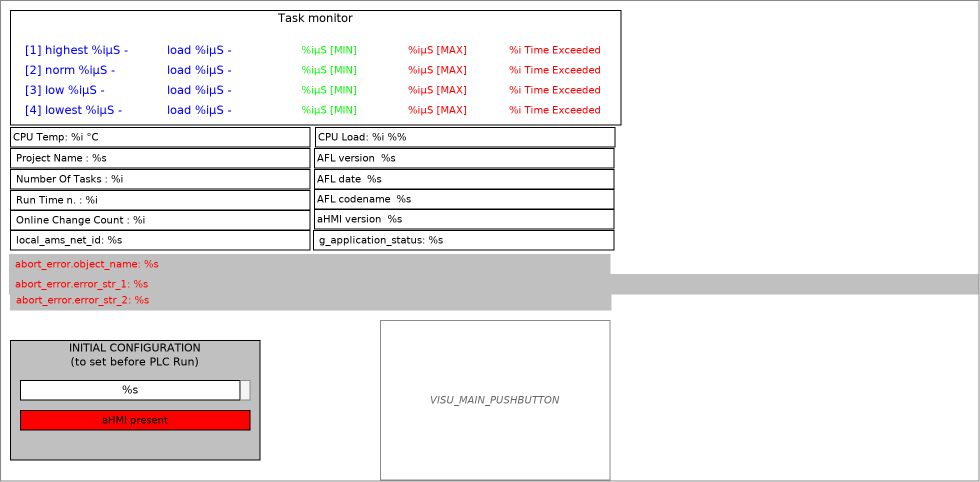
VISUALIZATION VISU_MAIN  // 980x482
    Rectangle (10,10 611x115), "Task monitor"
    Rectangle (9,254 601x20), "abort_error.object_name: %s", text variable: abort_error.object_name
    Rectangle (9,274 969x20), "abort_error.error_str_1: %s", text variable: abort_error.error_str_1
    Rectangle (10,290 601x20), "abort_error.error_str_2: %s", text variable: abort_error.error_str_2
    Rectangle (10,230 300x20), "local_ams_net_id: %s", text variable: local_ams_net_id
    Rectangle (313,230 301x20), "g_application_status: %s", text variable: Application_Common.g_application_status
    Rectangle (22,40 130x20), "[1] highest %iµS -", text variable: afl_tasks[1].cycle_us
    Rectangle (22,60 130x20), "[2] norm %iµS -", text variable: afl_tasks[2].cycle_us
    Rectangle (22,80 130x20), "[3] low %iµS -", text variable: afl_tasks[3].cycle_us
    Rectangle (22,100 130x20), "[4] lowest %iµS -", text variable: afl_tasks[4].cycle_us
    Rectangle (164,100 100x20), "load %iµS -", text variable: afl_tasks[4].task_profiler_data.AverageExecTime
    Rectangle (164,80 100x20), "load %iµS -", text variable: afl_tasks[3].task_profiler_data.AverageExecTime
    Rectangle (164,60 100x20), "load %iµS -", text variable: afl_tasks[2].task_profiler_data.AverageExecTime
    Rectangle (164,40 100x20), "load %iµS -", text variable: afl_tasks[1].task_profiler_data.AverageExecTime
    Rectangle (380,40 90x20), "%iµS [MAX]", text variable: afl_tasks[1].task_profiler_data.MaxExecTime
    Rectangle (380,60 90x20), "%iµS [MAX]", text variable: afl_tasks[2].task_profiler_data.MaxExecTime
    Rectangle (380,80 90x20), "%iµS [MAX]", text variable: afl_tasks[2].task_profiler_data.MaxExecTime
    Rectangle (380,100 90x20), "%iµS [MAX]", text variable: afl_tasks[4].task_profiler_data.MaxExecTime
    Rectangle (10,148 300x20), "Project Name : %s", text variable: SystemInfo.projectName
    Rectangle (10,169 300x20), "Number Of Tasks : %i", text variable: SystemInfo.numberOfTasks
    Rectangle (10,190 300x20), "Run Time n. : %i", text variable: SystemInfo.runTimeNo
    Rectangle (10,210 300x20), "Online Change Count : %i", text variable: SystemInfo.onlineChangeCount
    Rectangle (250,100 110x20), "%iµS [MIN]", text variable: afl_tasks[4].task_profiler_data.MinExecTime
    Rectangle (250,80 110x20), "%iµS [MIN]", text variable: afl_tasks[3].task_profiler_data.MinExecTime
    Rectangle (250,60 110x20), "%iµS [MIN]", text variable: afl_tasks[2].task_profiler_data.MinExecTime
    Rectangle (250,40 110x20), "%iµS [MIN]", text variable: afl_tasks[1].task_profiler_data.MinExecTime
    Rectangle (506,40 110x20), "%i Time Exceeded", text variable: SystemTaskInfoArr[1].cycleTimeExceeded
    Rectangle (506,60 110x20), "%i Time Exceeded", text variable: SystemTaskInfoArr[2].cycleTimeExceeded
    Rectangle (506,80 110x20), "%i Time Exceeded", text variable: SystemTaskInfoArr[3].cycleTimeExceeded
    Rectangle (506,100 110x20), "%i Time Exceeded", text variable: SystemTaskInfoArr[4].cycleTimeExceeded
    Rectangle (314,169 300x20), "AFL date %s", text variable: AFL_VERSION.v_date
    Rectangle (314,148 300x20), "AFL version %s", text variable: AFL_VERSION.s_value
    Rectangle (10,127 300x20), "CPU Temp: %i °C", text variable: .system_diagnosis.cpu_temperature_actual_value
    Rectangle (314,189 300x20), "AFL codename %s", text variable: AFL_VERSION.development_stage
    Rectangle (315,127 300x20), "CPU Load: %i %%", text variable: system_diagnosis.cpu_usage_actual_value
    Rectangle (314,209 300x20), "aHMI version %s", text variable: hmi.private.major_version
    Frame (380,320 230x160)
        shows VISU_MAIN_PUSHBUTTON(m_Input_mch := EZ.mch, m_Input_stop := ez_mch_services_pushbuttons_main.stop_button_di, m_Input_reset := ez_mch_services_pushbuttons_main.reset_button_di, m_Input_start := ez_mch_services_pushbuttons_main.start_button_pressed_di)
    Rectangle (10,340 250x120), "INITIAL CONFIGURATION (to set before PLC Run)", tooltip "selysionare la configurazione prima di mettere RUN il PLC"
    RoundedRectangle (20,410 230x20), "aHMI present", tooltip "Video presente e collegato", colour toggle: Application_Common.HMI_IS_REQUIRED_DVR
        toggle Application_Common.HMI_IS_REQUIRED_DVR
    RoundedRectangle (20,380 220x20), "%s", text variable: .test_target_device
    Scrollbar (240,380 10x20)
        p1057716461: .test_target_device
END_VISUALIZATION

(* stored: Version 1.1.0.1, ProductVersion 3.1.4024.3
   Visu VISU_MAIN: Id {0764160e-5c7c-421f-9d5a-5aa73c21b4bf} *)
